(* Logix 5000 project; controller SX_V040001_C001 vendor 1 type 14 code 77 rev 16.22; software revision 16.04; part 13 of 35 *)
(* tags used below, declared in another part *)
   ALL_KINDS : INT[90];
   DB_A_IO : INT[16];
   DB_D_IO : DINT[6];
   DB_D_IO_REVERSE : DINT[6];
   DRIVE : INT[32];
   EMPTYING : INT[18];
   G_AInput : DINT[8];
   G_DInput : DINT[3];
   G_DOutput : DINT[3];
   loading : INT[19];
   louvre : INT[11];
   m_alarm_exist : BOOL;
   m_on_off_line : BOOL;
   METERING : INT[44];
   PARAMETER : INT[501];
   REMOTE_SYSTEM : INT[38];
   STATUS_GENERAL : INT[135];
   STATUS_SEND_PART_1 : INT[135];
   TEMP : INT[14];
(* MainProgram, continued *)

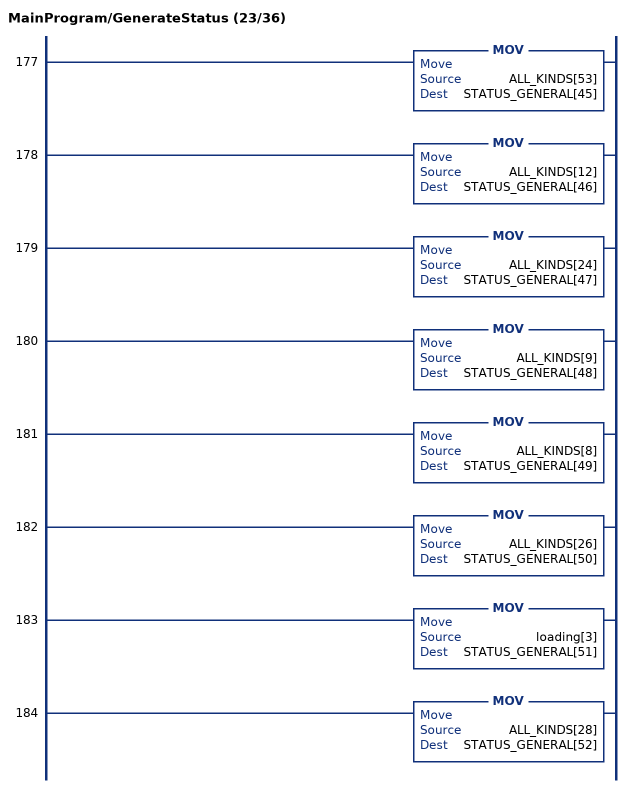
   [picture p284: MainProgram/GenerateStatus rungs 177-184]
   177: MOV(ALL_KINDS[53],STATUS_GENERAL[45]);
   178: MOV(ALL_KINDS[12],STATUS_GENERAL[46]);
   179: MOV(ALL_KINDS[24],STATUS_GENERAL[47]);
   180: MOV(ALL_KINDS[9],STATUS_GENERAL[48]);
   181: MOV(ALL_KINDS[8],STATUS_GENERAL[49]);
   182: MOV(ALL_KINDS[26],STATUS_GENERAL[50]);
   183: MOV(loading[3],STATUS_GENERAL[51]);
   184: MOV(ALL_KINDS[28],STATUS_GENERAL[52]);
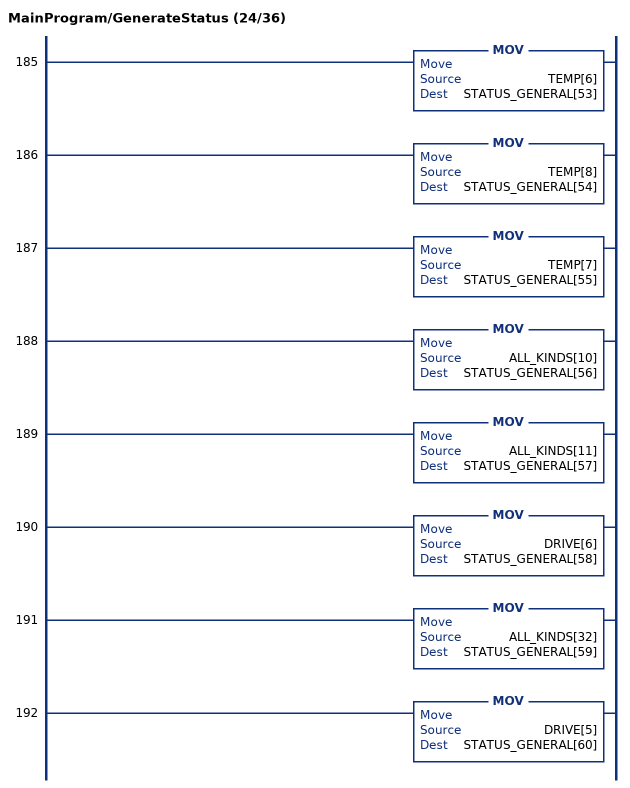
   185: MOV(TEMP[6],STATUS_GENERAL[53]);
   186: MOV(TEMP[8],STATUS_GENERAL[54]);
   187: MOV(TEMP[7],STATUS_GENERAL[55]);
   188: MOV(ALL_KINDS[10],STATUS_GENERAL[56]);
   189: MOV(ALL_KINDS[11],STATUS_GENERAL[57]);
   190: MOV(DRIVE[6],STATUS_GENERAL[58]);
   191: MOV(ALL_KINDS[32],STATUS_GENERAL[59]);
   192: MOV(DRIVE[5],STATUS_GENERAL[60]);
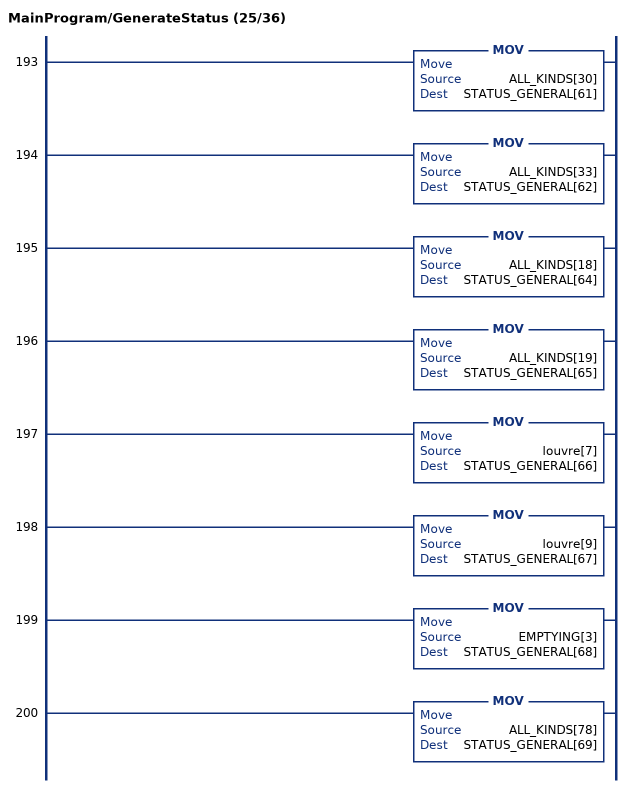
   193: MOV(ALL_KINDS[30],STATUS_GENERAL[61]);
   194: MOV(ALL_KINDS[33],STATUS_GENERAL[62]);
   195: MOV(ALL_KINDS[18],STATUS_GENERAL[64]);
   196: MOV(ALL_KINDS[19],STATUS_GENERAL[65]);
   197: MOV(louvre[7],STATUS_GENERAL[66]);
   198: MOV(louvre[9],STATUS_GENERAL[67]);
   199: MOV(EMPTYING[3],STATUS_GENERAL[68]);
   200: MOV(ALL_KINDS[78],STATUS_GENERAL[69]);
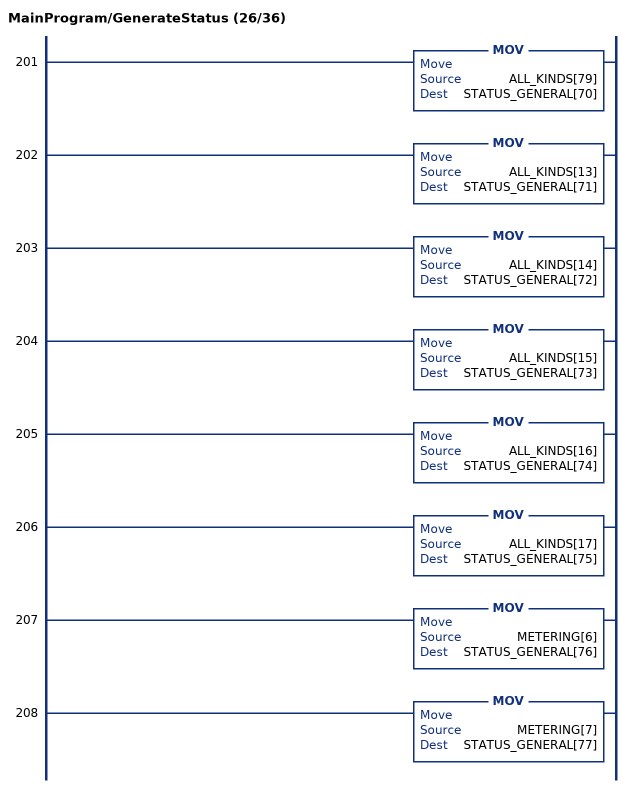
   201: MOV(ALL_KINDS[79],STATUS_GENERAL[70]);
   202: MOV(ALL_KINDS[13],STATUS_GENERAL[71]);
   203: MOV(ALL_KINDS[14],STATUS_GENERAL[72]);
   204: MOV(ALL_KINDS[15],STATUS_GENERAL[73]);
   205: MOV(ALL_KINDS[16],STATUS_GENERAL[74]);
   206: MOV(ALL_KINDS[17],STATUS_GENERAL[75]);
   207: MOV(METERING[6],STATUS_GENERAL[76]);
   208: MOV(METERING[7],STATUS_GENERAL[77]);
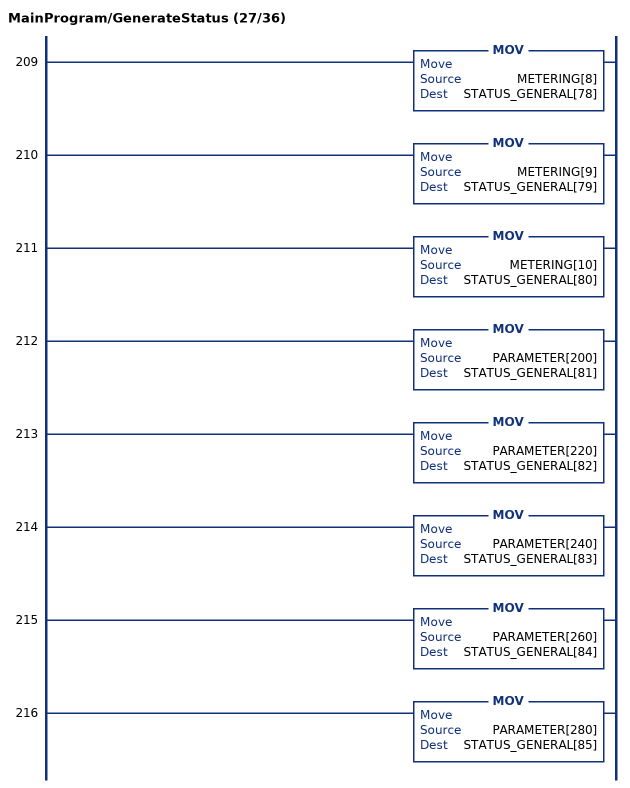
   209: MOV(METERING[8],STATUS_GENERAL[78]);
   210: MOV(METERING[9],STATUS_GENERAL[79]);
   211: MOV(METERING[10],STATUS_GENERAL[80]);
   212: MOV(PARAMETER[200],STATUS_GENERAL[81]);
   213: MOV(PARAMETER[220],STATUS_GENERAL[82]);
   214: MOV(PARAMETER[240],STATUS_GENERAL[83]);
   215: MOV(PARAMETER[260],STATUS_GENERAL[84]);
   216: MOV(PARAMETER[280],STATUS_GENERAL[85]);
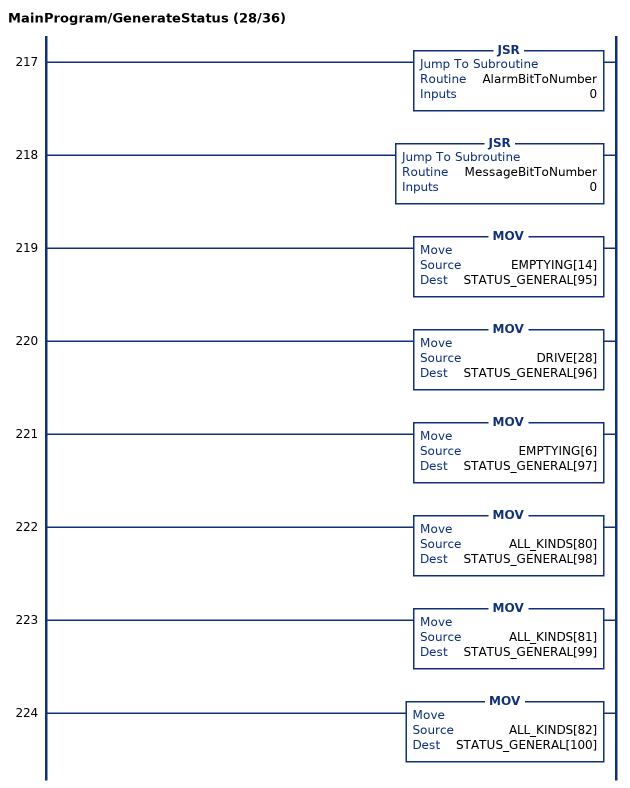
   217: JSR(AlarmBitToNumber,0);
   218: JSR(MessageBitToNumber,0);
   219: MOV(EMPTYING[14],STATUS_GENERAL[95]);
   220: MOV(DRIVE[28],STATUS_GENERAL[96]);
   221: MOV(EMPTYING[6],STATUS_GENERAL[97]);
   222: MOV(ALL_KINDS[80],STATUS_GENERAL[98]);
   223: MOV(ALL_KINDS[81],STATUS_GENERAL[99]);
   224: MOV(ALL_KINDS[82],STATUS_GENERAL[100]);
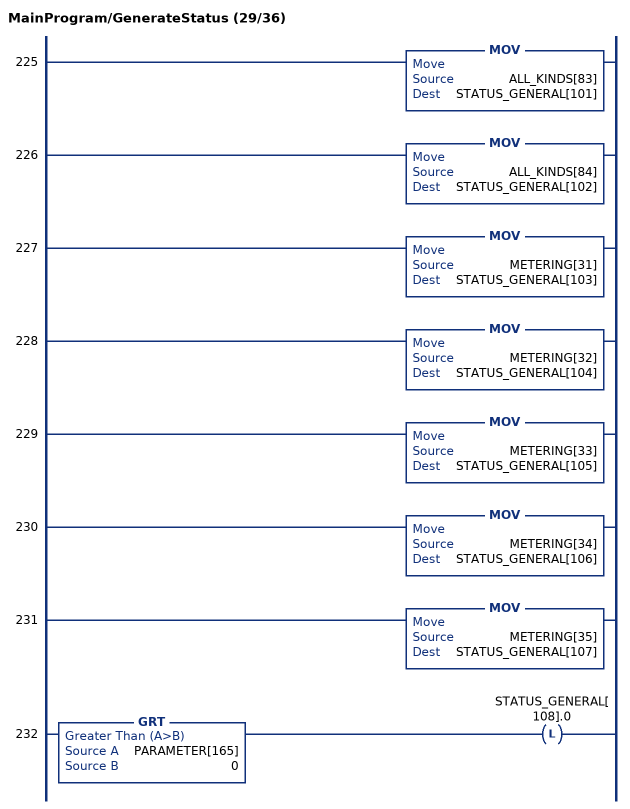
   225: MOV(ALL_KINDS[83],STATUS_GENERAL[101]);
   226: MOV(ALL_KINDS[84],STATUS_GENERAL[102]);
   227: MOV(METERING[31],STATUS_GENERAL[103]);
   228: MOV(METERING[32],STATUS_GENERAL[104]);
   229: MOV(METERING[33],STATUS_GENERAL[105]);
   230: MOV(METERING[34],STATUS_GENERAL[106]);
   231: MOV(METERING[35],STATUS_GENERAL[107]);
   232: GRT(PARAMETER[165],0)OTL(STATUS_GENERAL[108].0);
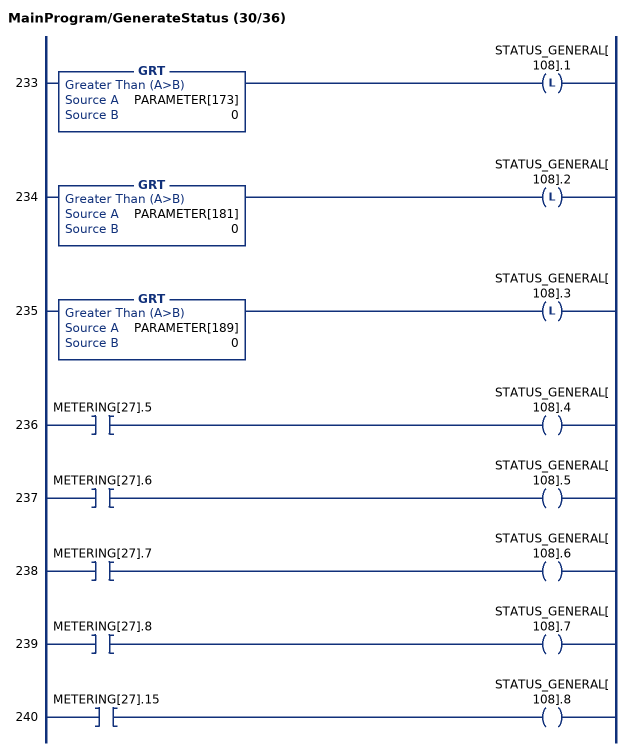
   233: GRT(PARAMETER[173],0)OTL(STATUS_GENERAL[108].1);
   234: GRT(PARAMETER[181],0)OTL(STATUS_GENERAL[108].2);
   235: GRT(PARAMETER[189],0)OTL(STATUS_GENERAL[108].3);
   236: XIC(METERING[27].5)OTE(STATUS_GENERAL[108].4);
   237: XIC(METERING[27].6)OTE(STATUS_GENERAL[108].5);
   238: XIC(METERING[27].7)OTE(STATUS_GENERAL[108].6);
   239: XIC(METERING[27].8)OTE(STATUS_GENERAL[108].7);
   240: XIC(METERING[27].15)OTE(STATUS_GENERAL[108].8);
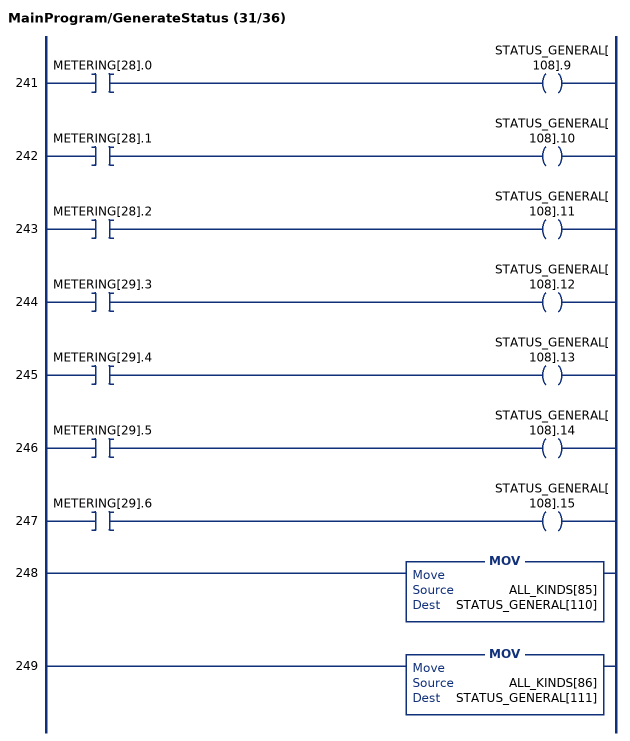
   241: XIC(METERING[28].0)OTE(STATUS_GENERAL[108].9);
   242: XIC(METERING[28].1)OTE(STATUS_GENERAL[108].10);
   243: XIC(METERING[28].2)OTE(STATUS_GENERAL[108].11);
   244: XIC(METERING[29].3)OTE(STATUS_GENERAL[108].12);
   245: XIC(METERING[29].4)OTE(STATUS_GENERAL[108].13);
   246: XIC(METERING[29].5)OTE(STATUS_GENERAL[108].14);
   247: XIC(METERING[29].6)OTE(STATUS_GENERAL[108].15);
   248: MOV(ALL_KINDS[85],STATUS_GENERAL[110]);
   249: MOV(ALL_KINDS[86],STATUS_GENERAL[111]);
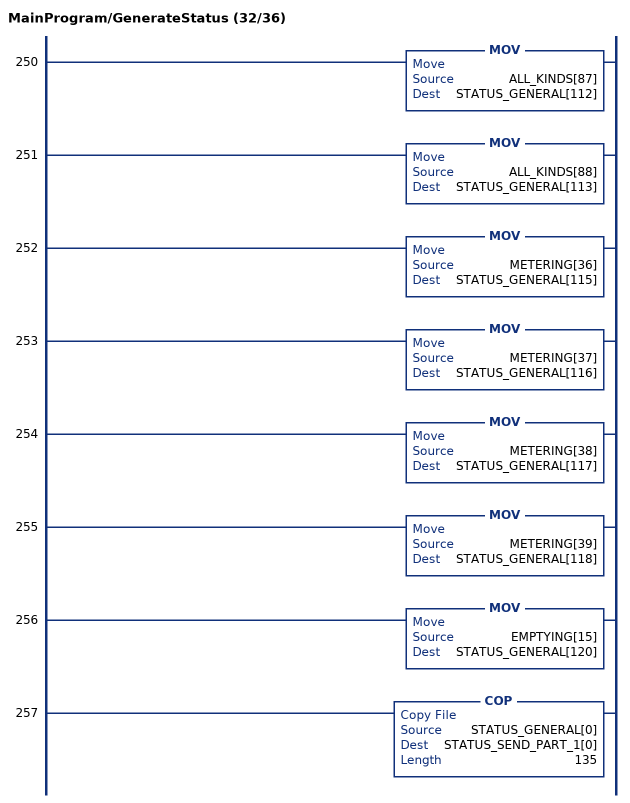
   250: MOV(ALL_KINDS[87],STATUS_GENERAL[112]);
   251: MOV(ALL_KINDS[88],STATUS_GENERAL[113]);
   252: MOV(METERING[36],STATUS_GENERAL[115]);
   253: MOV(METERING[37],STATUS_GENERAL[116]);
   254: MOV(METERING[38],STATUS_GENERAL[117]);
   255: MOV(METERING[39],STATUS_GENERAL[118]);
   256: MOV(EMPTYING[15],STATUS_GENERAL[120]);
   257: COP(STATUS_GENERAL[0],STATUS_SEND_PART_1[0],135);
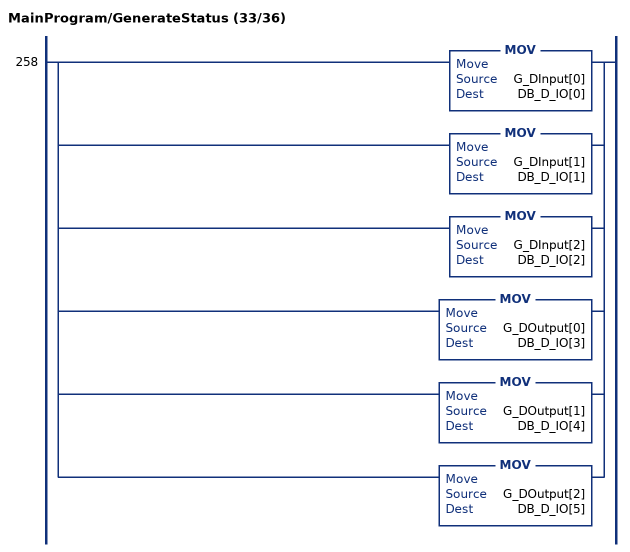
   258: [MOV(G_DInput[0],DB_D_IO[0]) ,MOV(G_DInput[1],DB_D_IO[1]) ,MOV(G_DInput[2],DB_D_IO[2]) ,MOV(G_DOutput[0],DB_D_IO[3]) ,MOV(G_DOutput[1],DB_D_IO[4]) ,MOV(G_DOutput[2],DB_D_IO[5]) ];
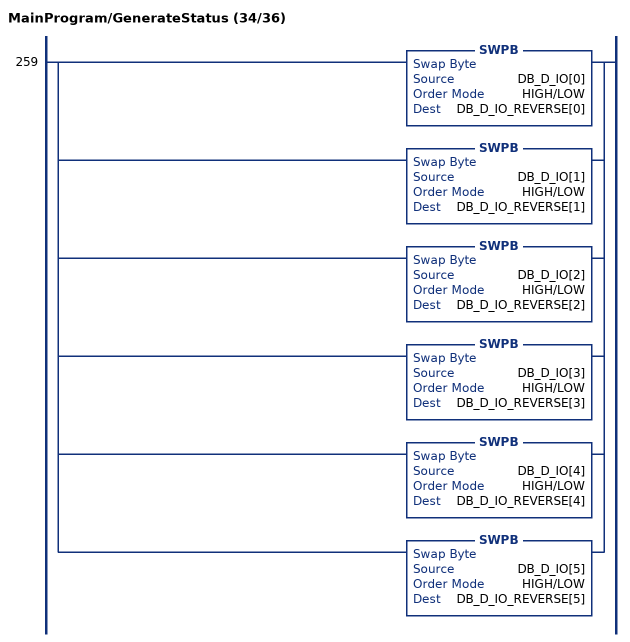
   259: [SWPB(DB_D_IO[0],HIGH/LOW,DB_D_IO_REVERSE[0]) ,SWPB(DB_D_IO[1],HIGH/LOW,DB_D_IO_REVERSE[1]) ,SWPB(DB_D_IO[2],HIGH/LOW,DB_D_IO_REVERSE[2]) ,SWPB(DB_D_IO[3],HIGH/LOW,DB_D_IO_REVERSE[3]) ,SWPB(DB_D_IO[4],HIGH/LOW,DB_D_IO_REVERSE[4]) ,SWPB(DB_D_IO[5],HIGH/LOW,DB_D_IO_REVERSE[5]) ];
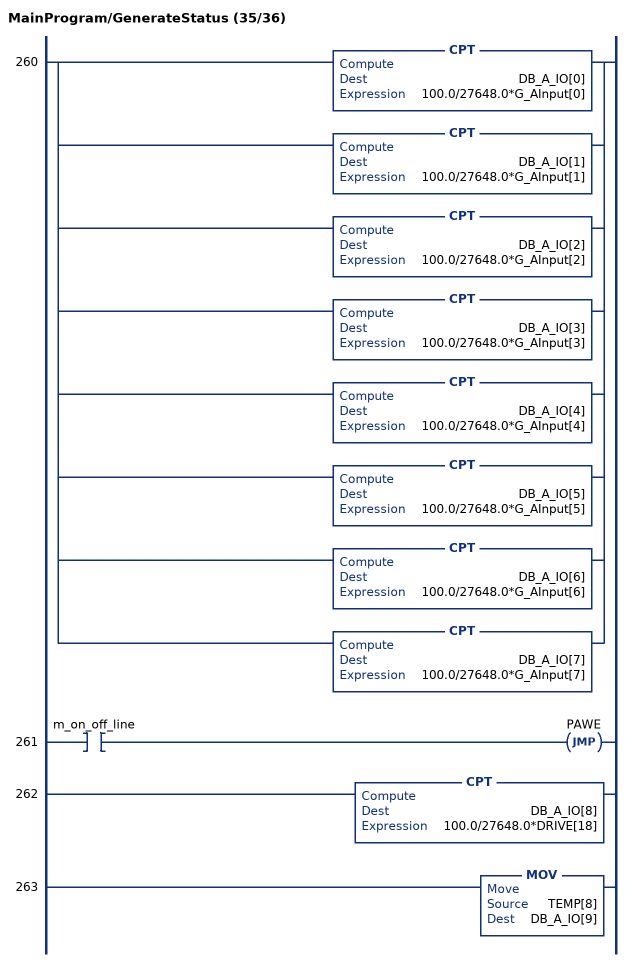
   260: [CPT(DB_A_IO[0],100.0/27648.0*G_AInput[0]) ,CPT(DB_A_IO[1],100.0/27648.0*G_AInput[1]) ,CPT(DB_A_IO[2],100.0/27648.0*G_AInput[2]) ,CPT(DB_A_IO[3],100.0/27648.0*G_AInput[3]) ,CPT(DB_A_IO[4],100.0/27648.0*G_AInput[4]) ,CPT(DB_A_IO[5],100.0/27648.0*G_AInput[5]) ,CPT(DB_A_IO[6],100.0/27648.0*G_AInput[6]) ,CPT(DB_A_IO[7],100.0/27648.0*G_AInput[7]) ];
   261: XIC(m_on_off_line)JMP(PAWE);
   262: CPT(DB_A_IO[8],100.0/27648.0*DRIVE[18]);
   263: MOV(TEMP[8],DB_A_IO[9]);
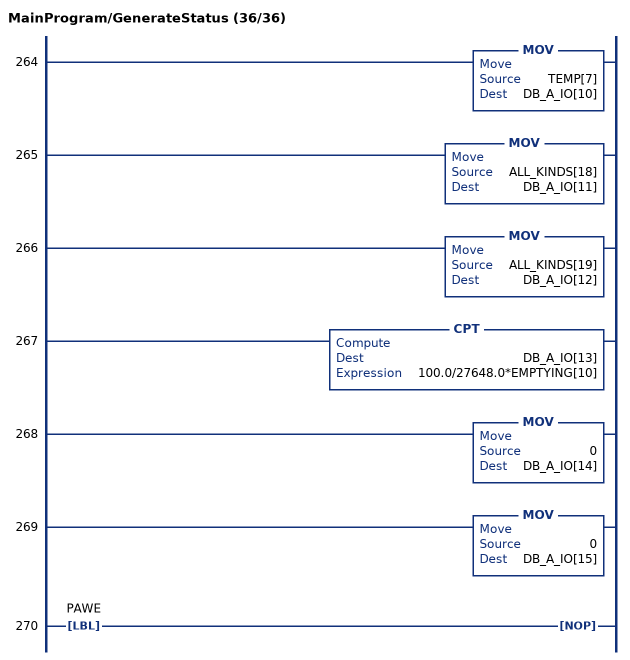
   264: MOV(TEMP[7],DB_A_IO[10]);
   265: MOV(ALL_KINDS[18],DB_A_IO[11]);
   266: MOV(ALL_KINDS[19],DB_A_IO[12]);
   267: CPT(DB_A_IO[13],100.0/27648.0*EMPTYING[10]);
   268: MOV(0,DB_A_IO[14]);
   269: MOV(0,DB_A_IO[15]);
   270: LBL(PAWE)NOP();
END_ROUTINE

ROUTINE GenStatusRM   (* ladder *)
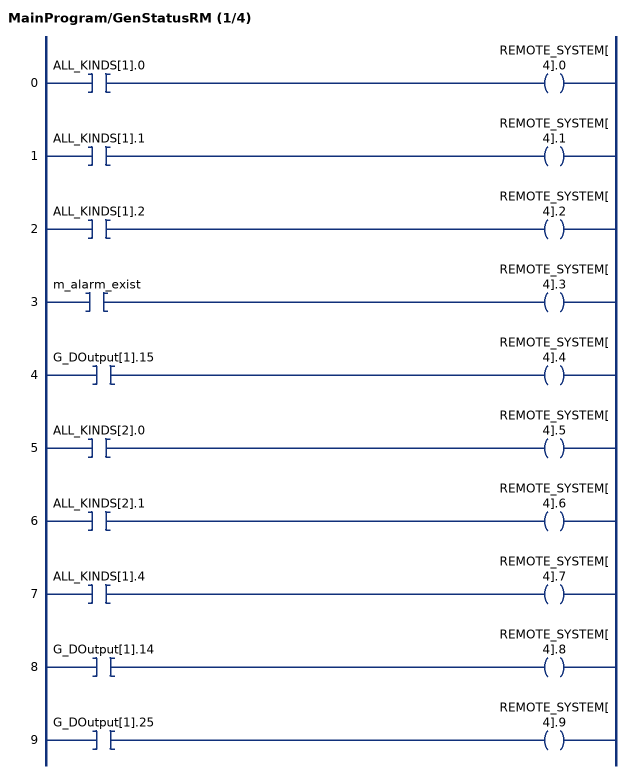
   0: XIC(ALL_KINDS[1].0)OTE(REMOTE_SYSTEM[4].0);
   1: XIC(ALL_KINDS[1].1)OTE(REMOTE_SYSTEM[4].1);
   2: XIC(ALL_KINDS[1].2)OTE(REMOTE_SYSTEM[4].2);
   3: XIC(m_alarm_exist)OTE(REMOTE_SYSTEM[4].3);
   4: XIC(G_DOutput[1].15)OTE(REMOTE_SYSTEM[4].4);
   5: XIC(ALL_KINDS[2].0)OTE(REMOTE_SYSTEM[4].5);
   6: XIC(ALL_KINDS[2].1)OTE(REMOTE_SYSTEM[4].6);
   7: XIC(ALL_KINDS[1].4)OTE(REMOTE_SYSTEM[4].7);
   8: XIC(G_DOutput[1].14)OTE(REMOTE_SYSTEM[4].8);
   9: XIC(G_DOutput[1].25)OTE(REMOTE_SYSTEM[4].9);
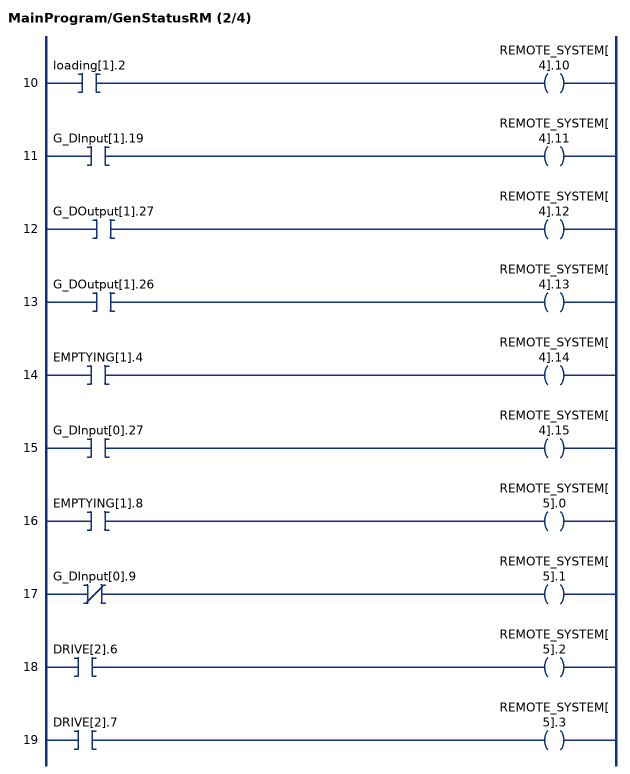
   10: XIC(loading[1].2)OTE(REMOTE_SYSTEM[4].10);
   11: XIC(G_DInput[1].19)OTE(REMOTE_SYSTEM[4].11);
   12: XIC(G_DOutput[1].27)OTE(REMOTE_SYSTEM[4].12);
   13: XIC(G_DOutput[1].26)OTE(REMOTE_SYSTEM[4].13);
   14: XIC(EMPTYING[1].4)OTE(REMOTE_SYSTEM[4].14);
   15: XIC(G_DInput[0].27)OTE(REMOTE_SYSTEM[4].15);
   16: XIC(EMPTYING[1].8)OTE(REMOTE_SYSTEM[5].0);
   17: XIO(G_DInput[0].9)OTE(REMOTE_SYSTEM[5].1);
   18: XIC(DRIVE[2].6)OTE(REMOTE_SYSTEM[5].2);
   19: XIC(DRIVE[2].7)OTE(REMOTE_SYSTEM[5].3);
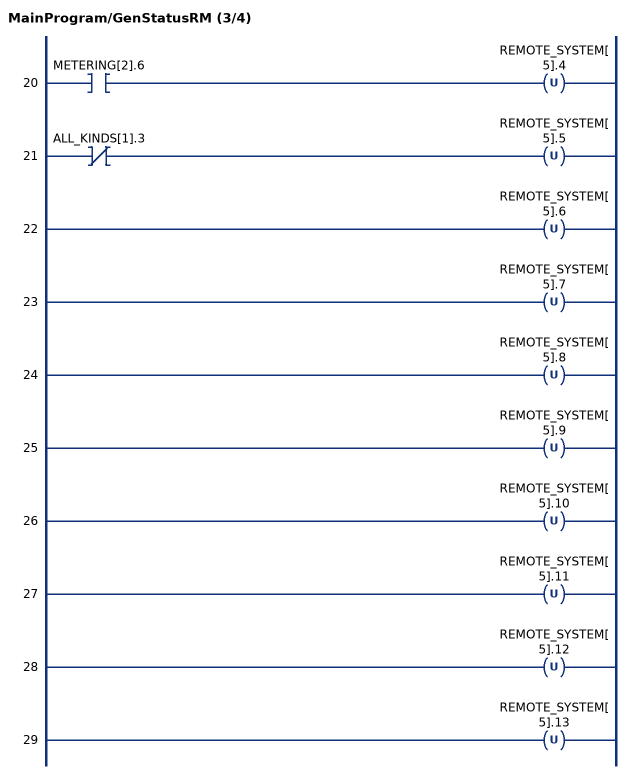
   20: XIC(METERING[2].6)OTU(REMOTE_SYSTEM[5].4);
   21: XIO(ALL_KINDS[1].3)OTU(REMOTE_SYSTEM[5].5);
   22: OTU(REMOTE_SYSTEM[5].6);
   23: OTU(REMOTE_SYSTEM[5].7);
   24: OTU(REMOTE_SYSTEM[5].8);
   25: OTU(REMOTE_SYSTEM[5].9);
   26: OTU(REMOTE_SYSTEM[5].10);
   27: OTU(REMOTE_SYSTEM[5].11);
   28: OTU(REMOTE_SYSTEM[5].12);
   29: OTU(REMOTE_SYSTEM[5].13);
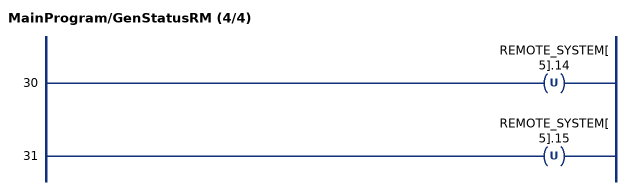
   30: OTU(REMOTE_SYSTEM[5].14);
   31: OTU(REMOTE_SYSTEM[5].15);
END_ROUTINE
